Staubli VAL3: libSignals.pjx

--- libSignals.pjx ---
Parameters version=s7.9.1 stackSize=5000 millimeterUnit=true
Program file=SA.pgx
Program file=SE.pgx
Program file=advMovesEmpty.pgx
Program file=avaAdvMoveIndex.pgx
Program file=blink.pgx
Program file=checkAdvMoves.pgx
Program file=destroyAdvMoves.pgx
Program file=exeBlink.pgx
Program file=exeMove_pulseDO.pgx
Program file=exeMove_setDO.pgx
Program file=exePulse.pgx
Program file=exeSA.pgx
Program file=exeSE.pgx
Program file=exeSearchL.pgx
Program file=exeSzone.pgx
Program file=exeWZone.pgx
Program file=freeAdvMove.pgx
Program file=killBlink.pgx
Program file=launchIdWD.pgx
Program file=lockAdvMove.pgx
Program file=MoveIdWatchdog.pgx
Program file=movej_pulseDO.pgx
Program file=movej_setDO.pgx
Program file=movel_pulseDO.pgx
Program file=movel_setDO.pgx
Program file=pulse.pgx
Program file=sZone.pgx
Program file=searchL.pgx
Program file=wZone.pgx
Data file=libSignals.dtx

--- libSignals.dtx ---
bool bSearchLFail
bool bSearchLSuccess
num nBlendOffToll = 0.1
num nBlendOnToll = 0.5
num nMaxTask = 10
num nMovesCount
num nPulseCount
num nSA_Count
num nSE_Count
num nSzoneCount
num nWzoneCount
bool bAdvMoveBusy[20]
string sAdvMovePrefix = "advMove"
bool bAdvMoves
string VERSION = "0.3.2"
num nDeadLockTout = 0.2

--- advMovesEmpty.pgx ---
program advMovesEmpty(bool& x_bRes)
  local num l_nIndex
begin

  //return true if the advanced moves stack is empty
  x_bRes=true
  for l_nIndex=0 to size(bAdvMoveBusy)-1
    if bAdvMoveBusy[l_nIndex]
      x_bRes=false
      return
    endIf
  endFor


end

--- avaAdvMoveIndex.pgx ---
program avaAdvMoveIndex(num& x_nIndex)
  local num l_nIndex
begin

  //return the first available "advanced move" index...-1 if max moves reached
  for l_nIndex=0 to size(bAdvMoveBusy)-1
    if !bAdvMoveBusy[l_nIndex]
      x_nIndex=l_nIndex
      return
    endIf
  endFor
  x_nIndex=-1

end

--- blink.pgx ---
public program blink(string x_sDioName, num x_nInterval, dio x_dDio)
begin

  //blink the output x_dDio with period x_nInterval

  if taskStatus("blink_"+x_sDioName)==-1
    taskCreate "blink_"+x_sDioName,10,exeBlink(x_dDio,x_nInterval)
    wait(taskStatus("blink_"+x_sDioName)==1)
  else
    //logMsg("libSignals/blink->can't create the blink task")
  endIf


end

--- checkAdvMoves.pgx ---
program checkAdvMoves()
  local num l_nIndex
begin

  //setMutex(bAdvMoves)
  for l_nIndex=0 to size(bAdvMoveBusy)-1
    if bAdvMoveBusy[l_nIndex]
      if taskStatus(sAdvMovePrefix+toString("",l_nIndex))==-1
        bAdvMoveBusy[l_nIndex]=false
      endIf
    endIf
  endFor
  //bAdvMoves=false

end

--- destroyAdvMoves.pgx ---
program destroyAdvMoves()
  local num l_nIndex
begin

  //setMutex(bAdvMoves)
  for l_nIndex=0 to size(bAdvMoveBusy)-1
    if bAdvMoveBusy[l_nIndex]
      taskKill(sAdvMovePrefix+toString("",l_nIndex))
      wait(taskStatus(sAdvMovePrefix+toString("",l_nIndex))==-1)
      bAdvMoveBusy[l_nIndex]=false
    endIf
  endFor
  //bAdvMoves=false

end

--- exeBlink.pgx ---
program exeBlink(dio x_dDio, num x_nInterval)
begin

  while true

    x_dDio=true
    delay(x_nInterval)
    x_dDio=false
    delay(x_nInterval)

  endWhile

end

--- exeMove_pulseDO.pgx ---
program exeMove_pulseDO(num x_nAdvMoveIndex, num x_nMoveId, point x_pPoint, tool x_tTool, num x_nDistance, num x_nPulseLength, dio x_dDio)
  local num l_givenId
  local num l_nDistance
  local num l_nMoveId
begin

  //I want to see the tool entering the zone
  //so at first I must be out
  wait(distance(position(here(x_tTool,world),world),position(x_pPoint,world))>=x_nDistance or roundDown(getMoveId())>roundDown(x_nMoveId))
  //then I go inside
  wait((distance(position(here(x_tTool,world),world),position(x_pPoint,world))<x_nDistance and roundDown(getMoveId())==roundDown(x_nMoveId)) or roundDown(getMoveId())>roundDown(x_nMoveId))

  if distance(position(here(x_tTool,world),world),position(x_pPoint,world))<x_nDistance
    //logMsg("libSignals/exeMove_PulseDO->success")
    call pulse(x_dDio,x_nPulseLength)
  elseIf roundDown(getMoveId())>roundDown(x_nMoveId)
    //the tool never passed close enough to x_pPoint
    logMsg("libSignals/exeMove_PulseDO->fail")
  endIf

  call freeAdvMove(x_nAdvMoveIndex)

end

--- exeMove_setDO.pgx ---
program exeMove_setDO(num x_nAdvMoveIndex, num x_nMoveId, point x_pPoint, tool x_tTool, num x_nDistance, dio x_dDio)
begin

  //I want to see the tool entering the zone
  //so at first I must be out
  wait(distance(position(here(x_tTool,world),world),position(x_pPoint,world))>=x_nDistance or roundDown(getMoveId())>roundDown(x_nMoveId))
  //then I go inside
  wait((distance(position(here(x_tTool,world),world),position(x_pPoint,world))<x_nDistance and roundDown(getMoveId())==roundDown(x_nMoveId)) or roundDown(getMoveId())>roundDown(x_nMoveId))

  if distance(position(here(x_tTool,world),world),position(x_pPoint,world))<x_nDistance
    //logMsg("libSignals/exeMove_SetDO->success")
    x_dDio=true
  elseIf roundDown(getMoveId())>roundDown(x_nMoveId)
    //the tool never passed close enough to x_pPoint
    logMsg("libSignals/exeMove_SetDO->fail")
  endIf

  call freeAdvMove(x_nAdvMoveIndex)

end

--- exePulse.pgx ---
program exePulse(dio x_dDio, num x_nLength)
begin

  //pulse execution

  x_dDio=true
  delay(x_nLength)
  x_dDio=false

end

--- exeSA.pgx ---
program exeSA(dio x_dInput, dio x_dOutput, num x_nLength)
begin

  while true
    x_dOutput=true
    wait(x_dInput==false)
    if (!watch(x_dInput==true,x_nLength))
      x_dOutput=false
    endIf
    wait(x_dInput==true)
    x_dOutput=true
  endWhile
end

--- exeSE.pgx ---
program exeSE(dio x_dInput, dio x_dOutput, num x_nLength)
begin

  while true
    x_dOutput=false
    wait(x_dInput==true)
    if !watch(x_dInput==false,x_nLength)
      x_dOutput=true
    endIf
    wait(x_dInput==false)
    x_dOutput=false
  endWhile

end

--- exeSearchL.pgx ---
program exeSearchL(dio x_dInput, tool x_tTool)
begin

  wait(x_dInput==true or bSearchLFail)
  if x_dInput==true
    resetMotion()
    bSearchLSuccess=true
  else
    logMsg("libSignals/exeSearchL->timeout")
  endIf

end

--- exeSzone.pgx ---
program exeSzone(tool x_tTool, point x_pPoint, frame x_fFrame, num x_Dx, num x_Dy, num x_Dz)
  local bool l_bXok
  local bool l_bYok
  local bool l_bZok
  local point l_pHere
begin
  while true
    l_pHere=here(x_tTool,x_fFrame)
    l_bXok=l_pHere.trsf.x>x_pPoint.trsf.x-x_Dx/2 and l_pHere.trsf.x<x_pPoint.trsf.x+x_Dx/2
    l_bYok=l_pHere.trsf.y>x_pPoint.trsf.y-x_Dy/2 and l_pHere.trsf.y<x_pPoint.trsf.y+x_Dy/2
    l_bZok=l_pHere.trsf.z>x_pPoint.trsf.z-x_Dz/2 and l_pHere.trsf.z<x_pPoint.trsf.z+x_Dz/2
    if (l_bXok and l_bYok and l_bZok)
      restartMove()
    else
      if workingMode()==3 or workingMode()==4 and isPowered()
        logMsg("libSignals/exeSZone->robot out of safe zone!")
        stopMove()
        disablePower()
      endIf
    endIf
    delay(0)
  endWhile
end

--- exeWZone.pgx ---
program exeWzone(tool x_tTool, point x_pPoint, frame x_fFrame, num x_Dx, num x_Dy, num x_Dz, dio x_dOut)
  local bool l_bXok
  local bool l_bYok
  local bool l_bZok
  local point l_pHere
begin
  while true
    l_pHere=here(x_tTool,x_fFrame)
    l_bXok=l_pHere.trsf.x>x_pPoint.trsf.x-x_Dx/2 and l_pHere.trsf.x<x_pPoint.trsf.x+x_Dx/2
    l_bYok=l_pHere.trsf.y>x_pPoint.trsf.y-x_Dy/2 and l_pHere.trsf.y<x_pPoint.trsf.y+x_Dy/2
    l_bZok=l_pHere.trsf.z>x_pPoint.trsf.z-x_Dz/2 and l_pHere.trsf.z<x_pPoint.trsf.z+x_Dz/2
    if l_bXok and l_bYok and l_bZok
      x_dOut=false
    else
      x_dOut=true
    endIf
    delay(0)
  endWhile
end

--- freeAdvMove.pgx ---
program freeAdvMove(num x_nIndex)
begin
  //setMutex(bAdvMoves)
  bAdvMoveBusy[x_nIndex]=false
  //bAdvMoves=false
end

--- killBlink.pgx ---
public program killBlink(string x_sDioName)
begin


  //destroy the task that is making the dio blinking...
  taskKill("blink_"+x_sDioName)
  wait(taskStatus("blink_"+x_sDioName)==-1)


end

--- launchIdWD.pgx ---
program launchIdWD()
begin

  //if not existing launch moveid watchdog task
  if taskStatus("moveIdWatchdog")!=1
    taskKill("moveIdWatchdog")
    wait(taskStatus("moveIdWatchdog")==-1)
    taskCreate "moveIdWatchdog",10,moveIdWatchdog()
    wait(taskStatus("moveIdWatchdog")==1)
  endIf

end

--- lockAdvMove.pgx ---
program lockAdvMove(num x_nIndex)
begin
  //setMutex(bAdvMoves)
  bAdvMoveBusy[x_nIndex]=true
  //bAdvMoves=false
end

--- MoveIdWatchdog.pgx ---
public program moveIdWatchdog()
  local bool l_bLoop
  local num l_nCurrMoveId
  local num l_nIndex
  local num l_nLastMoveId
  local string l_sTemp
  local bool l_bStackWasPop
begin

  //this program run as task can detect moveId alteration...sure there must be a better way to do it...
  //note:
  //      - it doesn't detect a setMoveId if it cause a moveId change < = 1
  //      - is done this way and not on the mere difference beacuse for some reason, sometime the moveId seems having a +-1 discontinuity for a single cicle...
  //        (see SRC-893)

  l_nLastMoveId=getMoveId()
  l_bLoop=true

  while l_bLoop

    l_nCurrMoveId=getMoveId()

    if (roundDown(l_nCurrMoveId)>roundDown(l_nLastMoveId)+1) or (roundDown(l_nCurrMoveId)<roundDown(l_nLastMoveId)-1) or (l_bStackWasPop and isEmpty())
      //resetMotion or SetMoveId detected!
      logMsg("libSignals/moveIdWatchdog->resetMotion or SetMoveId detected")
      setMutex(bAdvMoves)
      call destroyAdvMoves()
      bAdvMoves=false
    endIf

    l_nLastMoveId=l_nCurrMoveId
    //save if the movement stack was populated
    l_bStackWasPop=!isEmpty()

    //if possible kill the moveid watchdog task
    l_bLoop=false
    for l_nIndex=0 to size(bAdvMoveBusy)-1
      l_bLoop=l_bLoop or bAdvMoveBusy[l_nIndex]
    endFor

    delay(0)
  endWhile

end

--- movej_pulseDO.pgx ---
public program movej_pulseDO(point x_pPoint, tool x_tTool, mdesc x_mMdesc, dio& x_dDio, num x_nPulseLength)
  local bool l_bFound
  local num l_nDist
  local num l_nIndex
  local num l_nMoveId
  local bool l_bRes
begin

  //execute a movej with the usual arguments (x_pPoint, x_tTool, x_mMdesc) meanwhile
  //when the distance between x_tTool and x_pPoint is lesser than x_nDistance the output x_dDio produce an output of x_nPulseLength seconds

  //the stack is busy
  if bAdvMoves
    l_bRes = watch(!bAdvMoves, nDeadLockTout)
    if !l_bRes
      //it seems stuck!
      //check the "stack" compliance
      call checkAdvMoves()
      call advMovesEmpty(l_bRes)
      if l_bRes
        //but the stack is empty...someone changed it to true manually and saved the library?
        bAdvMoves = false
        libSave()
        logMsg("libSignals/movej_pulseDO->deadlock fixed")
      endIf
    endIf
  endIf

  setMutex(bAdvMoves)

  if x_mMdesc.blend==off
    l_nDist=nBlendOffToll
  else
    l_nDist=x_mMdesc.leave+nBlendOnToll
  endIf

  //check the "stack" compliance
  call checkAdvMoves()

  //get the first index available
  l_nIndex=-1
  while l_nIndex<0
    call avaAdvMoveIndex(l_nIndex)
    delay(0)
  endWhile

  if taskStatus(sAdvMovePrefix+toString("",l_nIndex))==-1
    call lockAdvMove(l_nIndex)
    taskCreate sAdvMovePrefix+toString("",l_nIndex),10,exeMove_pulseDO(l_nIndex, movej(x_pPoint,x_tTool,x_mMdesc),x_pPoint,x_tTool,l_nDist,x_nPulseLength,x_dDio)
    wait(taskStatus(sAdvMovePrefix+toString("",l_nIndex))==1)
    //launch id watchdog
    call launchIdWD()
  else
    logMsg("libSignals/movej_pulseDO->error creating the control task")
  endIf

  bAdvMoves = false

end

--- movej_setDO.pgx ---
public program movej_setDO(point x_pPoint, tool x_tTool, mdesc x_mMdesc, dio& x_dDio)
  local num l_nDist
  local num l_nIndex
  local bool l_bRes
begin

  //execute a movej with the usual arguments (x_pPoint, x_tTool, x_mMdesc) meanwhile
  //when the distance between x_tTool and x_pPoint is lesser than x_nDistance the output x_dDio is set to true

  //the stack is busy
  if bAdvMoves
    l_bRes = watch(!bAdvMoves, nDeadLockTout)
    if !l_bRes
      //it seems stuck!
      call advMovesEmpty(l_bRes)
      //check the "stack" compliance
      call checkAdvMoves()
      if l_bRes
        //but the stack is empty...someone changed it to true manually and saved the library?
        bAdvMoves = false
        libSave()
        logMsg("libSignals/movej_setDO->deadlock fixed")
      endIf
    endIf
  endIf

  setMutex(bAdvMoves)

  if x_mMdesc.blend==off
    l_nDist=nBlendOffToll
  else
    l_nDist=x_mMdesc.leave+nBlendOnToll
  endIf

  //check the "stack" compliance
  call checkAdvMoves()

  //get the first index available
  l_nIndex=-1
  while l_nIndex<0
    call avaAdvMoveIndex(l_nIndex)
    delay(0)
  endWhile

  if taskStatus(sAdvMovePrefix+toString("",l_nIndex))==-1
    call lockAdvMove(l_nIndex)
    taskCreate sAdvMovePrefix+toString("",l_nIndex),10,exeMove_setDO(l_nIndex, movej(x_pPoint,x_tTool,x_mMdesc),x_pPoint,x_tTool,l_nDist,x_dDio)
    wait(taskStatus(sAdvMovePrefix+toString("",l_nIndex))==1)
    //launch id watchdog
    call launchIdWD()
  else
    logMsg("libSignals/movej_setDO->error creating the control task")
  endIf

  bAdvMoves = false


end

--- movel_pulseDO.pgx ---
public program movel_pulseDO(point x_pPoint, tool x_tTool, mdesc x_mMdesc, dio& x_dDio, num x_nPulseLength)
  local num l_nDist
  local num l_nIndex
  local bool l_bRes
begin

  //execute a movel with the usual arguments (x_pPoint, x_tTool, x_mMdesc) meanwhile
  //when the distance between x_tTool and x_pPoint is lesser than x_nDistance the output x_dDio produce an output of x_nPulseLength seconds

  //the stack is busy
  if bAdvMoves
    l_bRes = watch(!bAdvMoves, nDeadLockTout)
    if !l_bRes
      //it seems stuck!
      call advMovesEmpty(l_bRes)
      //check the "stack" compliance
      call checkAdvMoves()
      if l_bRes
        //but the stack is empty...someone changed it to true manually and saved the library?
        bAdvMoves = false
        libSave()
        logMsg("libSignals/movel_pulseDO->deadlock fixed")
      endIf
    endIf
  endIf

  setMutex(bAdvMoves)

  if x_mMdesc.blend==off
    l_nDist=nBlendOffToll
  else
    l_nDist=x_mMdesc.leave+nBlendOnToll
  endIf

  //check the "stack" compliance
  call checkAdvMoves()

  //get the first index available
  l_nIndex=-1
  while l_nIndex<0
    call avaAdvMoveIndex(l_nIndex)
    delay(0)
  endWhile

  if taskStatus(sAdvMovePrefix+toString("",l_nIndex))==-1
    call lockAdvMove(l_nIndex)
    taskCreate sAdvMovePrefix+toString("",l_nIndex),10,exeMove_pulseDO(l_nIndex, movel(x_pPoint,x_tTool,x_mMdesc),x_pPoint,x_tTool,l_nDist,x_nPulseLength,x_dDio)
    //launch id watchdog
    call launchIdWD()
  else
    logMsg("libSignals/movel_pulseDO->error creating the control task")
  endIf

  bAdvMoves = false


end

--- movel_setDO.pgx ---
public program movel_setDO(point x_pPoint, tool x_tTool, mdesc x_mMdesc, dio& x_dDio)
  local num l_nDist
  local num l_nIndex
  local bool l_bRes
begin

  //execute a movej with the usual arguments (x_pPoint, x_tTool, x_mMdesc) meanwhile
  //when the distance between x_tTool and x_pPoint is lesser than x_nDistance the output x_dDio is set to true

  //the stack is busy
  if bAdvMoves
    l_bRes = watch(!bAdvMoves, nDeadLockTout)
    if !l_bRes
      //it seems stuck!
      call advMovesEmpty(l_bRes)
      //check the "stack" compliance
      call checkAdvMoves()
      if l_bRes
        //but the stack is empty...someone changed it to true manually and saved the library?
        bAdvMoves = false
        libSave()
        logMsg("libSignals/movel_setDO->deadlock fixed")
      endIf
    endIf
  endIf

  setMutex(bAdvMoves)

  if x_mMdesc.blend==off
    l_nDist=nBlendOffToll
  else
    l_nDist=x_mMdesc.leave+nBlendOnToll
  endIf

  //check the "stack" compliance
  call checkAdvMoves()

  //get the first index available
  l_nIndex=-1
  while l_nIndex<0
    call avaAdvMoveIndex(l_nIndex)
    delay(0)
  endWhile

  //get the first index available
  l_nIndex=-1
  while l_nIndex<0
    call avaAdvMoveIndex(l_nIndex)
    delay(0)
  endWhile

  if taskStatus(sAdvMovePrefix+toString("",l_nIndex))==-1
    call lockAdvMove(l_nIndex)
    taskCreate sAdvMovePrefix+toString("",l_nIndex),10,exeMove_setDO(l_nIndex, movel(x_pPoint,x_tTool,x_mMdesc),x_pPoint,x_tTool,l_nDist,x_dDio)
    wait(taskStatus(sAdvMovePrefix+toString("",l_nIndex))==1)
    //launch id watchdog
    call launchIdWD()
  else
    logMsg("libSignals/movel_setDO->error creating the control task")
  endIf

  bAdvMoves = false


end

--- pulse.pgx ---
public program pulse(dio x_dDio, num x_nLength)
begin

  //generates a pulse of x_nLength for the output x_dDio

  if taskStatus("pulse_"+toString("",nPulseCount))==-1
    taskCreate "pulse_"+toString("",nPulseCount),10,exePulse(x_dDio,x_nLength)
    nPulseCount=nPulseCount+1
    if nPulseCount>nMaxTask
      nPulseCount=0
    endIf
  else
    logMsg("libSignals/pulse->can't create the task!")
  endIf

end

--- SA.pgx ---
public program SA(dio x_dInput, dio x_dOutput, num x_nLength)
begin

  //"reset delay"
  //reset the x_dOutput only when x_dInput is false for a time greater than x_nLength
  //note: x_dInput isn't necessarily an input

  if taskStatus("SA_"+toString("",nSA_Count))==-1
    taskCreate "SA_"+toString("",nSA_Count),10,exeSA(x_dInput,x_dOutput,x_nLength)
    nSA_Count=nSA_Count+1
    if nSA_Count>nMaxTask
      nSA_Count=0
    endIf
  else
    logMsg("libSignals/SA->can't create SA task")
  endIf

end

--- SE.pgx ---
public program SE(dio x_dInput, dio x_dOutput, num x_nLength)
begin

  //"set delay"
  //set the x_dOutput only when x_dInput is true for a time greater than x_nLength
  //note: x_dInput isn't necessarily an input

  if taskStatus("SE_"+toString("",nSE_Count))==-1
    taskCreate "SE_"+toString("",nSE_Count),10,exeSE(x_dInput,x_dOutput,x_nLength)
    nSE_Count=nSE_Count+1
    if nSE_Count>nMaxTask
      nSE_Count=0
    endIf
  else
    logMsg("libSignals/SE->can't create SE task")
  endIf

end

--- searchL.pgx ---
public program searchL(point x_pEndSearch, tool x_tTool, mdesc x_mMdesc, frame& x_fFrame, dio x_dInput, point& x_pFound)
  local mdesc l_mMdesc
begin

  //execute a movel from x_pStartSearch to x_pEndSearch
  //if x_dInput switch to true during this movement the robot stops and the current position of x_tTool is written in x_pFound
  //note: x_dInput isn't necessarily an input, the blend of the movement is set to off by default

  bSearchLFail=false
  bSearchLSuccess=false

  if taskStatus("searchL")==-1
    taskCreate "searchL",10,exeSearchL(x_dInput,x_tTool)
  else
    logMsg("libSignals/searchL->error creating the control task")
  endIf

  l_mMdesc=x_mMdesc
  l_mMdesc.blend=off

  movel(x_pEndSearch,x_tTool,l_mMdesc)
  wait(distance(here(x_tTool,x_fFrame),x_pEndSearch)<nBlendOffToll or bSearchLSuccess)
  if !bSearchLSuccess
    bSearchLFail=true
  else
    x_pFound=here(x_tTool,x_fFrame)
  endIf
end

--- sZone.pgx ---
public program sZone(tool x_tTool, point x_pPoint, frame x_fFrame, num x_Dx, num x_Dy, num x_Dz)
begin

  //in automatic mode stop immediately the robot if x_tTool is out of a box defined as:

  //x_pPoint.trsf.x + x_Dx/2 > here(x_tTool, x_fFrame).x > x_pPoint.trsf.x - x_Dx/2
  //x_pPoint.trsf.y + x_Dy/2 > here(x_tTool, x_fFrame).y > x_pPoint.trsf.y - x_Dy/2
  //x_pPoint.trsf.z + x_Dz/2 > here(x_tTool, x_fFrame).z > x_pPoint.trsf.z - x_Dz/2

  if taskStatus("sZone_"+toString("",nSzoneCount))==-1
    taskCreate "sZone_"+toString("",nSzoneCount),15,exeSzone(x_tTool,x_pPoint,x_fFrame,x_Dx,x_Dy,x_Dz)
    nSzoneCount=nSzoneCount+1
    if nSzoneCount>nMaxTask
      nSzoneCount=0
    endIf
  else
    logMsg("libSignals/sZone->can't create the task")
  endIf

end

--- wZone.pgx ---
public program wZone(tool x_tTool, point x_pPoint, frame x_fFrame, num x_Dx, num x_Dy, num x_Dz, dio& x_dOut)
begin

  //set x_dOut to false if x_tTool is inside a box defined as:

  //x_pPoint.trsf.x + x_Dx/2 > here(x_tTool, x_fFrame).x > x_pPoint.trsf.x - x_Dx/2
  //x_pPoint.trsf.y + x_Dy/2 > here(x_tTool, x_fFrame).y > x_pPoint.trsf.y - x_Dy/2
  //x_pPoint.trsf.z + x_Dz/2 > here(x_tTool, x_fFrame).z > x_pPoint.trsf.z - x_Dz/2

  if taskStatus("wZone_"+toString("",nWzoneCount))==-1
    taskCreate "wZone_"+toString("",nWzoneCount),15,exeWzone(x_tTool,x_pPoint,x_fFrame,x_Dx,x_Dy,x_Dz,x_dOut)
    nWzoneCount=nWzoneCount+1
    if nWzoneCount>nMaxTask
      nWzoneCount=0
    endIf
  else
    logMsg("libSignals/wZone->can't create the task")
  endIf


end
